// TIA Portal V20 export
TYPE "LKinCtrl_typeDiagnosticsPathSelect"
TITLE = typeDiagnosticsFBTemplate
   STRUCT
      status : Word;   // Status of the FC or error identification when error occurred
      entryID : Int;   // identifier for false entry
   END_STRUCT;
END_TYPE
